// TIA Portal project "Parking_Project_With_Hmi" (V16)

(* hardware
DEVICE "S7-1200 station_1"  S7-1200 Station
   slot 0: "Rack_0"  S7-1200 Rack  Rack  V1.0
   slot 1: "PLC_1"  CPU 1212C DC/DC/DC  6ES7 212-1AE40-0XB0  V4.4
DEVICE "HMI_1"  TP700 Comfort
   slot 0: "HMI_1"  TP700 Comfort  6AV2 124-0GC01-0AX0  16.0.0.0
   slot 1: "HMI_RT_1"  TP700 Comfort  6AV2 124-0GC01-0AX0  16.0.0.0
   slot 5: "HMI_1.IE_CP_1"  PROFINET Interface  16.0.0.0
      slot 1: "PROFINET Interface_1"  PROFINET Interface
         slot 1: "Port_1"  Port
         slot 2: "Port_2"  Port
   slot 7: "HMI_1.MPI/DP_CP_1"  MPI/DP Interface  16.0.0.0
*)

// ===== PLC "PLC_1"  CPU 1212C DC/DC/DC =====

VAR_GLOBAL   // PLC tag table "Default tag table"
   "START" AT %M0.0 : Bool;
   "STOP" AT %M0.1 : Bool;
   "RESET" AT %M0.2 : Bool;
   "ENTRY_SENSOR" AT %M0.3 : Bool;
   "EXIT_SENSOR" AT %M0.4 : Bool;
   "LOAD" AT %M0.5 : Bool;
   "ENTRY_GATE_OPENING" AT %M0.6 : Bool;
   "ENTRY_GATE_HOLD" AT %M0.7 : Bool;
   "ENTRY_GATE_CLOSING" AT %M1.0 : Bool;
   "EXIT_GATE_OPENING" AT %M1.1 : Bool;
   "EXIT_GATE_HOLD" AT %M1.2 : Bool;
   "EXIT_GATE_CLOSING" AT %M1.3 : Bool;
   "PARKING_FULL" AT %M1.4 : Bool;
   "PARKING_EMPTY" AT %M1.5 : Bool;
   "TOTAL_PARKING" AT %MW10 : Word;
   "AVAILABLE_PARKING" AT %MW20 : Word;
   "OCCUPIED_PARKING" AT %MW30 : Word;
   "USE_ENTRY_RED" AT %M3.5 : Bool;
   "USE_EXIT_RED" AT %M3.6 : Bool;
END_VAR

DATA_BLOCK "ALARM"   // DB1
{ S7_Optimized_Access := 'FALSE' }
VERSION : 0.1
   VAR
      ALARM : Struct
         ENTRY_GATE_OPENING : Bool;
         ENTRY_GATE_OPEN : Bool;
         ENTRY_GATE_CLOSING : Bool;
         ENTRY_GATE_CLOSE : Bool;
         EXIT_GATE_CLOSE : Bool;
         EXIT_GATE_OPENING : Bool;
         EXIT_GATE_CLOSING : Bool;
         EXIT_GATE_OPEN : Bool;
      END_STRUCT;
   END_VAR
BEGIN
END_DATA_BLOCK

DATA_BLOCK "Parking_FB1"   // DB3
{ S7_Optimized_Access := 'TRUE' }
VERSION : 0.1
// stored: InstanceOfName Parking_FB
"Parking_FB"
BEGIN
END_DATA_BLOCK

FUNCTION_BLOCK "Parking_FB"   // FB1, LAD
{ S7_Optimized_Access := 'TRUE' }
VERSION : 0.1
   VAR_INPUT
      ENTRY_SENSOR : Bool;
      EXIT_SENSOR : Bool;
      RESET : Bool;
      LOAD : Bool;
      TOTAL_PARKING_SPACE : Word;
   END_VAR
   VAR_OUTPUT
      ENTRY_GATE_OPENING : Bool;
      ENTRY_GATE_HOLD : Bool;
      ENTRY_GATE_CLOSING : Bool;
      EXIT_GATE_OPENING : Bool;
      EXIT_GATE_HOLD : Bool;
      EXIT_GATE_CLOSING : Bool;
      OCCUPIED_PARKING_SPACE : Word;
      PARKING_FULL : Bool;
      PARKING_EMPTY : Bool;
      AVAILABLE_PARKING_SPACE : Word;
   END_VAR
   VAR RETAIN
      COUNTER1 : CTUD_INT;
   END_VAR
   VAR
      ENTRY_GATE_OPN : TP_TIME;
      ENTRY_GATE_HLD : TP_TIME;
      ENTRY_GATE_CLSING : TP_TIME;
      TIMEER : TP_TIME;
      EXIT_GATE_OPN : TP_TIME;
      EXIT_GATE_HLD : TP_TIME;
      EXIT_GATE_CLSING : TP_TIME;
   END_VAR
BEGIN

REGION Network 1
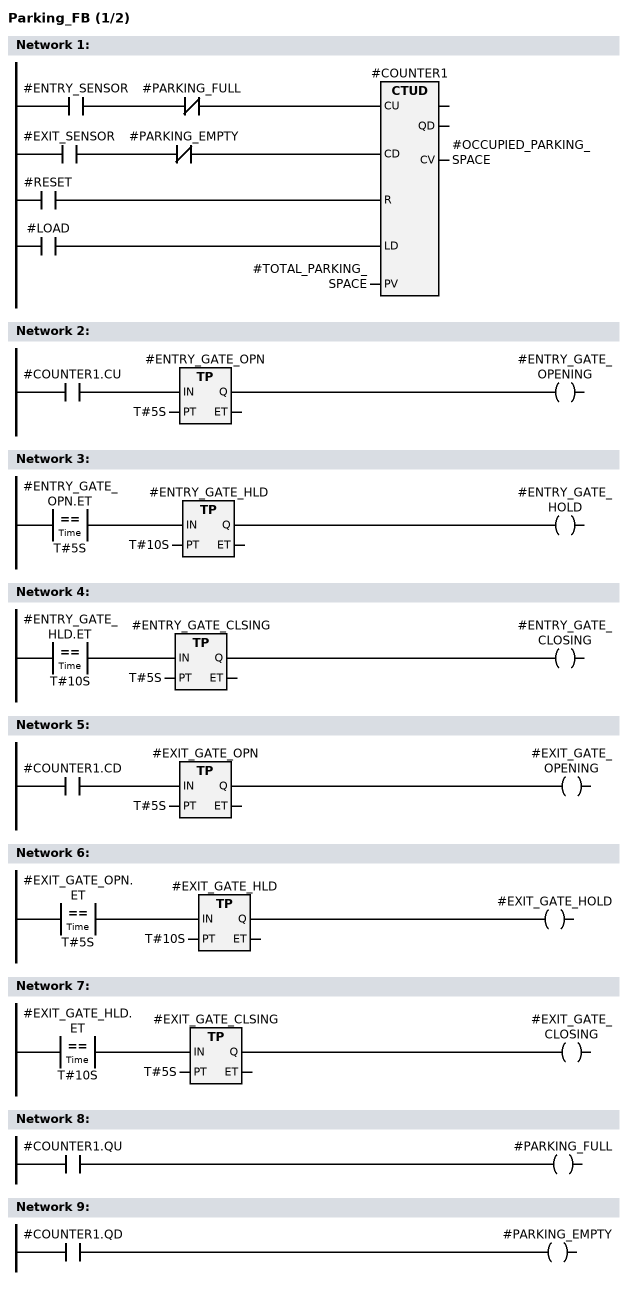
   #COUNTER1(CU := #ENTRY_SENSOR AND NOT #PARKING_FULL,   // CTUD
             CD := #EXIT_SENSOR AND NOT #PARKING_EMPTY,
             R := #RESET,
             LD := #LOAD,
             PV := #TOTAL_PARKING_SPACE,
             CV => #OCCUPIED_PARKING_SPACE);
END_REGION

REGION Network 2
   #ENTRY_GATE_OPN(IN := #COUNTER1.CU, PT := T#5S);   // TP
   #ENTRY_GATE_OPENING := #ENTRY_GATE_OPN.Q;
END_REGION

REGION Network 3
   #ENTRY_GATE_HLD(IN := #ENTRY_GATE_OPN.ET = T#5S, PT := T#10S);   // TP
   #ENTRY_GATE_HOLD := #ENTRY_GATE_HLD.Q;
END_REGION

REGION Network 4
   #ENTRY_GATE_CLSING(IN := #ENTRY_GATE_HLD.ET = T#10S, PT := T#5S);   // TP
   #ENTRY_GATE_CLOSING := #ENTRY_GATE_CLSING.Q;
END_REGION

REGION Network 5
   #EXIT_GATE_OPN(IN := #COUNTER1.CD, PT := T#5S);   // TP
   #EXIT_GATE_OPENING := #EXIT_GATE_OPN.Q;
END_REGION

REGION Network 6
   #EXIT_GATE_HLD(IN := #EXIT_GATE_OPN.ET = T#5S, PT := T#10S);   // TP
   #EXIT_GATE_HOLD := #EXIT_GATE_HLD.Q;
END_REGION

REGION Network 7
   #EXIT_GATE_CLSING(IN := #EXIT_GATE_HLD.ET = T#10S, PT := T#5S);   // TP
   #EXIT_GATE_CLOSING := #EXIT_GATE_CLSING.Q;
END_REGION

REGION Network 8
   RUNG wire#powerrail
      Contact( #COUNTER1.QU )
      Coil( #PARKING_FULL )
   END_RUNG
   // the same network as SCL:
   #PARKING_FULL := #COUNTER1.QU;
END_REGION

REGION Network 9
   RUNG wire#powerrail
      Contact( #COUNTER1.QD )
      Coil( #PARKING_EMPTY )
   END_RUNG
   // the same network as SCL:
   #PARKING_EMPTY := #COUNTER1.QD;
END_REGION

REGION Network 10
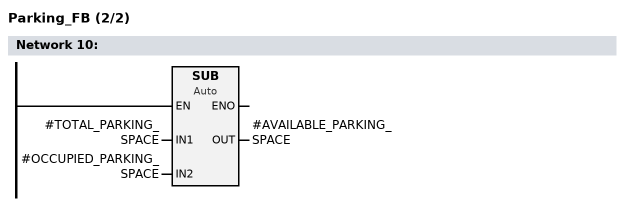
   RUNG wire#powerrail
      Sub(in1 := #TOTAL_PARKING_SPACE, in2 := #OCCUPIED_PARKING_SPACE, out => #AVAILABLE_PARKING_SPACE)
   END_RUNG
   // the same network as SCL:
   #AVAILABLE_PARKING_SPACE := #TOTAL_PARKING_SPACE - #OCCUPIED_PARKING_SPACE;
END_REGION
END_FUNCTION_BLOCK

ORGANIZATION_BLOCK "Main"   // OB1, LAD, ProgramCycle
TITLE = "Main Program Sweep (Cycle)"
{ S7_Optimized_Access := 'TRUE' }
VERSION : 0.1
   VAR_INPUT
      Initial_Call : Bool;   // Initial call of this OB
      Remanence : Bool;   // =True, if remanent data are available
   END_VAR
BEGIN

REGION Network 1
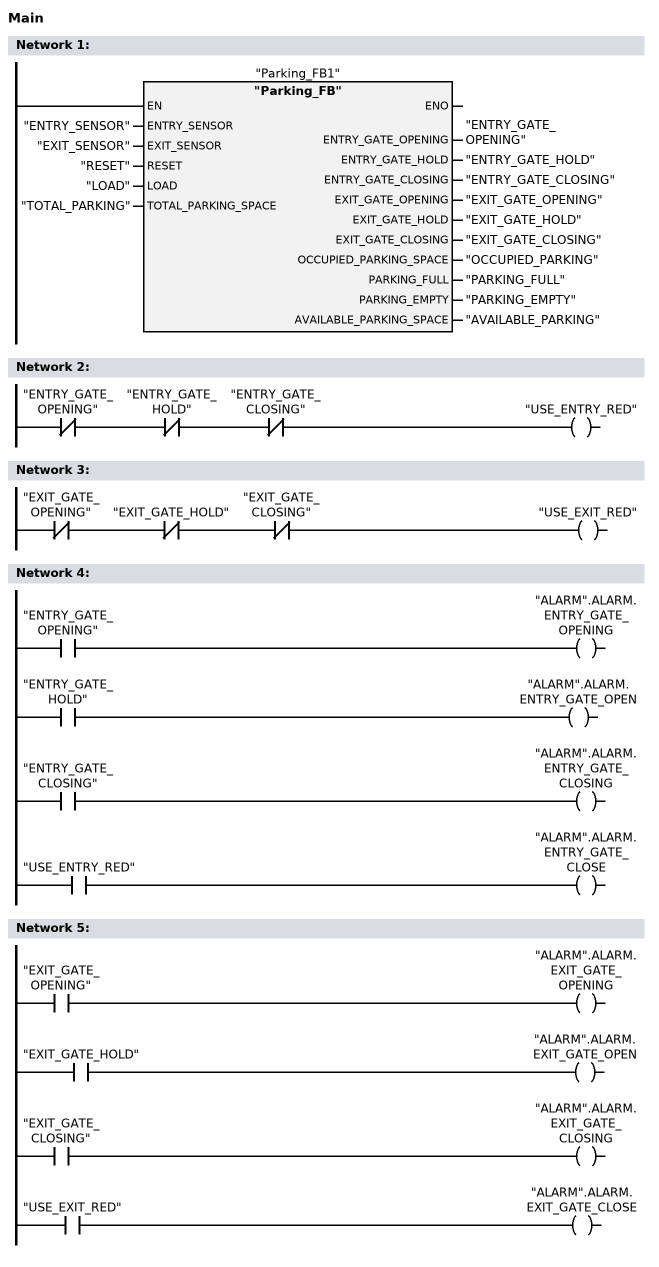
   RUNG wire#powerrail
      "Parking_FB1"(ENTRY_SENSOR := "ENTRY_SENSOR", EXIT_SENSOR := "EXIT_SENSOR", RESET := "RESET", LOAD := "LOAD", TOTAL_PARKING_SPACE := "TOTAL_PARKING", ENTRY_GATE_OPENING => "ENTRY_GATE_OPENING", ENTRY_GATE_HOLD => "ENTRY_GATE_HOLD", ENTRY_GATE_CLOSING => "ENTRY_GATE_CLOSING", EXIT_GATE_OPENING => "EXIT_GATE_OPENING", EXIT_GATE_HOLD => "EXIT_GATE_HOLD", EXIT_GATE_CLOSING => "EXIT_GATE_CLOSING", OCCUPIED_PARKING_SPACE => "OCCUPIED_PARKING", PARKING_FULL => "PARKING_FULL", PARKING_EMPTY => "PARKING_EMPTY", AVAILABLE_PARKING_SPACE => "AVAILABLE_PARKING")
   END_RUNG
   // the same network as SCL:
   "Parking_FB1"(ENTRY_SENSOR := "ENTRY_SENSOR",   // "Parking_FB"
                 EXIT_SENSOR := "EXIT_SENSOR",
                 RESET := "RESET",
                 LOAD := "LOAD",
                 TOTAL_PARKING_SPACE := "TOTAL_PARKING",
                 ENTRY_GATE_OPENING => "ENTRY_GATE_OPENING",
                 ENTRY_GATE_HOLD => "ENTRY_GATE_HOLD",
                 ENTRY_GATE_CLOSING => "ENTRY_GATE_CLOSING",
                 EXIT_GATE_OPENING => "EXIT_GATE_OPENING",
                 EXIT_GATE_HOLD => "EXIT_GATE_HOLD",
                 EXIT_GATE_CLOSING => "EXIT_GATE_CLOSING",
                 OCCUPIED_PARKING_SPACE => "OCCUPIED_PARKING",
                 PARKING_FULL => "PARKING_FULL",
                 PARKING_EMPTY => "PARKING_EMPTY",
                 AVAILABLE_PARKING_SPACE => "AVAILABLE_PARKING");
END_REGION

REGION Network 2
   RUNG wire#powerrail
      I_Contact( "ENTRY_GATE_OPENING" )
      I_Contact( "ENTRY_GATE_HOLD" )
      I_Contact( "ENTRY_GATE_CLOSING" )
      Coil( "USE_ENTRY_RED" )
   END_RUNG
   // the same network as SCL:
   "USE_ENTRY_RED" := NOT "ENTRY_GATE_OPENING" AND NOT "ENTRY_GATE_HOLD" AND NOT "ENTRY_GATE_CLOSING";
END_REGION

REGION Network 3
   RUNG wire#powerrail
      I_Contact( "EXIT_GATE_OPENING" )
      I_Contact( "EXIT_GATE_HOLD" )
      I_Contact( "EXIT_GATE_CLOSING" )
      Coil( "USE_EXIT_RED" )
   END_RUNG
   // the same network as SCL:
   "USE_EXIT_RED" := NOT "EXIT_GATE_OPENING" AND NOT "EXIT_GATE_HOLD" AND NOT "EXIT_GATE_CLOSING";
END_REGION

REGION Network 4
   RUNG wire#powerrail
      Contact( "ENTRY_GATE_OPENING" )
      Coil( "ALARM".ALARM.ENTRY_GATE_OPENING )
   END_RUNG
   RUNG wire#powerrail
      Contact( "ENTRY_GATE_HOLD" )
      Coil( "ALARM".ALARM.ENTRY_GATE_OPEN )
   END_RUNG
   RUNG wire#powerrail
      Contact( "ENTRY_GATE_CLOSING" )
      Coil( "ALARM".ALARM.ENTRY_GATE_CLOSING )
   END_RUNG
   RUNG wire#powerrail
      Contact( "USE_ENTRY_RED" )
      Coil( "ALARM".ALARM.ENTRY_GATE_CLOSE )
   END_RUNG
   // the same network as SCL:
   "ALARM".ALARM.ENTRY_GATE_OPENING := "ENTRY_GATE_OPENING";
   "ALARM".ALARM.ENTRY_GATE_OPEN := "ENTRY_GATE_HOLD";
   "ALARM".ALARM.ENTRY_GATE_CLOSING := "ENTRY_GATE_CLOSING";
   "ALARM".ALARM.ENTRY_GATE_CLOSE := "USE_ENTRY_RED";
END_REGION

REGION Network 5
   RUNG wire#powerrail
      Contact( "EXIT_GATE_OPENING" )
      Coil( "ALARM".ALARM.EXIT_GATE_OPENING )
   END_RUNG
   RUNG wire#powerrail
      Contact( "EXIT_GATE_HOLD" )
      Coil( "ALARM".ALARM.EXIT_GATE_OPEN )
   END_RUNG
   RUNG wire#powerrail
      Contact( "EXIT_GATE_CLOSING" )
      Coil( "ALARM".ALARM.EXIT_GATE_CLOSING )
   END_RUNG
   RUNG wire#powerrail
      Contact( "USE_EXIT_RED" )
      Coil( "ALARM".ALARM.EXIT_GATE_CLOSE )
   END_RUNG
   // the same network as SCL:
   "ALARM".ALARM.EXIT_GATE_OPENING := "EXIT_GATE_OPENING";
   "ALARM".ALARM.EXIT_GATE_OPEN := "EXIT_GATE_HOLD";
   "ALARM".ALARM.EXIT_GATE_CLOSING := "EXIT_GATE_CLOSING";
   "ALARM".ALARM.EXIT_GATE_CLOSE := "USE_EXIT_RED";
END_REGION
END_ORGANIZATION_BLOCK

(* ===== HMI "HMI_RT_1" =====
system functions are stored by id; their names below are inferred from use
connection "HMI_Connection_1": ETHERNET, S7_1200_OMS

HMI tags "Default tag table"
   "AVAILABLE_PARKING" : Word = PLC AVAILABLE_PARKING AT %MW20, 1 s
   "OCCUPIED_PARKING" : Word = PLC OCCUPIED_PARKING AT %MW30, 1 s
   "PARKING_FULL" : Bool = PLC PARKING_FULL AT %M1.4, 1 s
   "PARKING_EMPTY" : Bool = PLC PARKING_EMPTY AT %M1.5, 1 s
   "ENTRY_GATE_OPENING" : Bool = PLC ENTRY_GATE_OPENING AT %M0.6, 1 s
   "EXIT_GATE_OPENING" : Bool = PLC EXIT_GATE_OPENING AT %M1.1, 1 s
   "ENTRY_GATE_HOLD" : Bool = PLC ENTRY_GATE_HOLD AT %M0.7, 1 s
   "EXIT_GATE_HOLD" : Bool = PLC EXIT_GATE_HOLD AT %M1.2, 1 s
   "ENTRY_GATE_CLOSING" : Bool = PLC ENTRY_GATE_CLOSING AT %M1.0, 1 s
   "EXIT_GATE_CLOSING" : Bool = PLC EXIT_GATE_CLOSING AT %M1.3, 1 s
   "USE_ENTRY_RED" : Bool = PLC USE_ENTRY_RED AT %M3.5, 1 s
   "USE_EXIT_RED" : Bool = PLC USE_EXIT_RED AT %M3.6, 1 s
   "TOTAL_PARKING" : Word = PLC TOTAL_PARKING AT %MW10, 1 s
   "ENTRY_SENSOR" : Bool = PLC ENTRY_SENSOR AT %M0.3, 1 s
   "ALARM" : Int AT %DB1.DBW0, 1 s
   "EXIT_SENSOR" : Bool = PLC EXIT_SENSOR AT %M0.4, 1 s

discrete alarms
   1: 'ENTRY_GATE_CLOSE', class Errors, trigger "ALARM" bit 11
   3: 'ENTRY_GATE_OPEN', class Errors, trigger "ALARM" bit 9
   8: 'EXIT_GATE_CLOSING', class Errors, trigger "ALARM" bit 14
   7: 'EXIT_GATE_OPEN', class Errors, trigger "ALARM" bit 15
   6: 'EXIT_GATE_OPENING', class Errors, trigger "ALARM" bit 13
   2: 'ENTRY_GATE_OPENING', class Errors, trigger "ALARM" bit 8
   5: 'EXIT_GATE_CLOSE', class Errors, trigger "ALARM" bit 12
   4: 'ENTRY_GATE_CLOSING', class Errors, trigger "ALARM" bit 10

screen "Root screen" 800x480, template "Template_1"
   Button "Button_3" at 301,51 size 205x36; TextOff 'PARKING FULL'
      Visibility <- "PARKING_FULL"
   IOField "I/O field_1" at 461,294 size 92x43; FormatPattern 99999
      ProcessValue <- "AVAILABLE_PARKING"
   IOField "I/O field_2" at 461,207 size 90x42; FormatPattern 99999
      ProcessValue <- "OCCUPIED_PARKING"
   Button "Button_1" at 169,381 size 173x35; TextOff 'STATUS OF GATE'
      on Click: function_efd93a16("STATUS_OF_GATE", 0, 0, -1, -1, 1)
   IOField "I/O field_3" at 457,113 size 92x43; FormatPattern 99999
      ProcessValue <- "TOTAL_PARKING"
   Button "Button_4" at 301,52 size 206x35; TextOff 'PARKING EMPTY'
      Visibility <- "PARKING_EMPTY"
   Button "Button_5" at 166,114 size 243x42; TextOff 'TOTAL PARKING SPACE'
   Button "Button_6" at 166,207 size 243x42; TextOff 'OCCUPIED SPACE'
   Button "Button_7" at 166,297 size 243x42; TextOff 'AVAILABLE SPACE'
   Button "Button_2" at 411,381 size 96x35; TextOff 'UPDATES'
      on Click: ActivateScreen("ALARM_SCREEN", 0)

PopupScreen "STATUS_OF_GATE" 280x280
   TextField "Text field_1" at 70,24 size 66x23; Text 'ENTRY'
   TextField "Text field_2" at 185,25 size 48x23; Text 'EXIT'
   GraphicView "Graphic view_2" at 95,90 size 57x27; Picture "Graphic_2"
      Visibility <- "ENTRY_GATE_OPENING"
      Appearance <- "ENTRY_GATE_OPENING"
   GraphicView "Graphic view_6" at 179,88 size 60x28; Picture "Graphic_2"
      Visibility <- "EXIT_GATE_OPENING"
      Appearance <- "EXIT_GATE_OPENING"
   GraphicView "Graphic view_13" at 182,121 size 57x28; Picture "Graphic_2"
      Visibility <- "EXIT_GATE_HOLD"
      Appearance <- "EXIT_GATE_HOLD"
   GraphicView "Graphic view_8" at 91,124 size 59x29; Picture "Graphic_2"
      Visibility <- "ENTRY_GATE_HOLD"
      Appearance <- "ENTRY_GATE_HOLD"
   GraphicView "Graphic view_15" at 92,155 size 59x29; Picture "Graphic_2"
      Visibility <- "ENTRY_GATE_CLOSING"
      Appearance <- "ENTRY_GATE_CLOSING"
   GraphicView "Graphic view_18" at 182,154 size 57x30; Picture "Graphic_2"
      Appearance <- "EXIT_GATE_CLOSING"
      Visibility <- "EXIT_GATE_CLOSING"
   GraphicView "Graphic view_21" at 93,192 size 58x30; Picture "Graphic_2"
      Visibility <- "USE_ENTRY_RED"
      Appearance <- "USE_ENTRY_RED"
   GraphicView "Graphic view_24" at 182,192 size 57x30; Picture "Graphic_2"
      Visibility <- "USE_EXIT_RED"
      Appearance <- "USE_EXIT_RED"
   Button "Button_1" at 0,232 size 96x41; TextOff 'CLOSE'
      on Click: function_efd93a16("STATUS_OF_GATE", 0, 0, 0, -1, 1)
   TextField "Text field_3" at 76,48 size 54x23; Text 'GATE'
   TextField "Text field_4" at 179,47 size 54x23; Text 'GATE'
   TextField "Text field_5" at 0,165 size 83x22; Text 'CLOSING'
   TextField "Text field_6" at 4,198 size 72x22; Text 'CLOSED'
   TextField "Text field_7" at 25,132 size 52x22; Text 'OPEN'
   TextField "Text field_8" at 0,93 size 85x22; Text 'OPENING'

screen "ALARM_SCREEN" 800x480
   AlarmView "Alarm view_1" at 112,73 size 600x300
   Button "Button_1" at 58,413 size 114x35; TextOff 'WELCOME'
      on Click: ActivateScreen("Root screen", 0)
*)